(* PLC project Tc2_Utilities.F_GetWeekOfTheYear Demo, tc3-libraries-kb TwinCAT 3.1 *)
(* stored: creationDateTime 2026-05-10T12:00:00, modificationDateTime 2026-05-10T12:00:00 *)

PROGRAM P_Demo_F_GetWeekOfTheYear
  VAR
    rResult : WORD;  (* F_GetWeekOfTheYear 的返回值 *)
    bRun : BOOL;  (* 触发一次调用 *)
    dtNow : DATE_AND_TIME := DT#2008-03-17-12:00;  (* 测试用本地变量 *)
  END_VAR

            // ============================================================
// Tc2_Utilities.F_GetWeekOfTheYear 演示程序（FUNCTION）
// ============================================================
// 验证步骤：
//   1. 引用 Tc2_Utilities（及类型所在依赖库 Tc2_System / Tc2_Standard）
//   2. 编译 + 登录
//   3. 强制 bRun := TRUE 一个周期
//   4. 观察 rResult 应为 12
// ============================================================

IF bRun THEN
    rResult := F_GetWeekOfTheYear(dtNow);
    bRun := FALSE;
END_IF;

          
END_PROGRAM
